// TIA Portal V18 export
FUNCTION_BLOCK "FB_MES_Monitoring"   // FB4, SCL
{ S7_Optimized_Access := 'TRUE' }
// stored: IsIECCheckEnabled true, MemoryReserve 100, SetENOAutomatically false
   VAR_INPUT
      Enable : Bool := TRUE;
      Reset : Bool := FALSE;
      HeartbeatTimeout_MES : Time := T#6s;
      HeartbeatTimeout_PLC : Time := T#6s;
      CheckInTimeout : Time := T#10s;
      CheckOutTimeout : Time := T#10s;
      StoveCheckInTimeout : Time := T#10s;
   END_VAR
   VAR_IN_OUT
      Diag : "UDT_MES_Monitoring";
   END_VAR
   VAR
      _hbMesValue : Bool;
      _hbPlcValue : Bool;
      _errCode : Array[1..8] of DInt;
      _errText : Array[1..8] of String[128];
      _actErrIdx : Array[1..8] of Int;
      _actErrCnt : Int;
      _actErrPos : Int;
      _errRotateEnable : Bool;
      _tErrRotate { S7_SetPoint := 'True'} : TON_TIME;
      _hbMesLast : Bool;
      _hbPlcLast : Bool;
      _tHbMes { S7_SetPoint := 'True'} : TON_TIME;
      _tHbPlc { S7_SetPoint := 'True'} : TON_TIME;
      _tCi { S7_SetPoint := 'True'} : Array[1..8] of TON_TIME;
      _tCo { S7_SetPoint := 'True'} : Array[1..8] of TON_TIME;
      _tStove { S7_SetPoint := 'True'} : TON_TIME;
      _ciDonePrev : Array[1..8] of Bool;
      _coDonePrev : Array[1..8] of Bool;
      _ciOkPrev : Array[1..8] of Bool;
      _ciNgPrev : Array[1..8] of Bool;
      _coOkPrev : Array[1..8] of Bool;
      _coNgPrev : Array[1..8] of Bool;
      _ciTimeoutLatched : Array[1..8] of Bool;
      _coTimeoutLatched : Array[1..8] of Bool;
      _spDonePrev : Array[1..8] of Bool;
      _spOkPrev : Array[1..8] of Bool;
      _spNgPrev : Array[1..8] of Bool;
      _lrDonePrev : Array[1..8] of Bool;
      _lrOkPrev : Array[1..8] of Bool;
      _lrNgPrev : Array[1..8] of Bool;
      _stoveOkPrev : Bool;
      _stoveTimeoutLatched : Bool;
      _i : Int;
      _ciReq : Array[1..8] of Bool;
      _ciOk : Array[1..8] of Bool;
      _ciNg : Array[1..8] of Bool;
      _ciDone : Array[1..8] of Bool;
      _coReq : Array[1..8] of Bool;
      _coOk : Array[1..8] of Bool;
      _coNg : Array[1..8] of Bool;
      _coDone : Array[1..8] of Bool;
      _spOk : Array[1..8] of Bool;
      _spNg : Array[1..8] of Bool;
      _spDone : Array[1..8] of Bool;
      _lrOk : Array[1..8] of Bool;
      _lrNg : Array[1..8] of Bool;
      _lrDone : Array[1..8] of Bool;
      _stoveReq : Bool;
      _stoveOk : Bool;
   END_VAR
BEGIN
   (*
   ===============================================================================
   BLOCK / PURPOSE
   ===============================================================================
   This code builds a MES diagnostics snapshot (#Diag) from PLC<->MES handshake DBs.
   It:
   - Mirrors key signals into #Diag.Header / #Diag.LastError / #Diag.Special / #Diag.Station[i]
   - Measures heartbeat "age" and timeout for MES and PLC heartbeats
   - Tracks per-station handshake counters (OK / NG / Done / Timeout) with edge detection
   - Latches "UnexpectedDone" if Done arrives without active request
   - Implements RESET to clear all counters/flags in #Diag
   ===============================================================================
   ASSUMPTIONS / NOTES
   ===============================================================================
   - #_tHbMes, #_tHbPlc, #_tStove and #_tCi[], #_tCo[] are IEC TON timers
   - #HeartbeatTimeout_MES / _PLC, #CheckInTimeout, #CheckOutTimeout, #StoveCheckInTimeout are TIME
   - Indexing: stations are 1..8
   - "ChickIn" naming in tags is preserved as-is (typo likely in original DB)
   ===============================================================================
   *)

   REGION "GUARD / ENABLE"
     IF NOT #Enable THEN
       RETURN;
     END_IF;
   END_REGION

   REGION "READ RAW SIGNALS FROM DBs (PLC<->MES + LAST ERROR)"
     #_hbMesValue := "MEStoPLC"."MES.HeartbeatSignal";
     #_hbPlcValue := "PLCtoMES"."PLC.Unload_HeartbeatSignal";

     // Unload error per station
     #_errCode[1] := "Station1UnLoadData"."MES.ErrorCode";
     #_errText[1] := "Station1UnLoadData"."MES.ErrorMsg";

     #_errCode[2] := "Station2UnLoadData"."MES.ErrorCode";
     #_errText[2] := "Station2UnLoadData"."MES.ErrorMsg";

     #_errCode[3] := "Station3UnLoadData"."MES.ErrorCode";
     #_errText[3] := "Station3UnLoadData"."MES.ErrorMsg";

     #_errCode[4] := "Station4UnLoadData"."MES.ErrorCode";
     #_errText[4] := "Station4UnLoadData"."MES.ErrorMsg";

     #_errCode[5] := "Station5UnLoadData"."MES.ErrorCode";
     #_errText[5] := "Station5UnLoadData"."MES.ErrorMsg";

     #_errCode[6] := "Station6UnLoadData"."MES.ErrorCode";
     #_errText[6] := "Station6UnLoadData"."MES.ErrorMsg";

     #_errCode[7] := "Station7UnLoadData"."MES.ErrorCode";
     #_errText[7] := "Station7UnLoadData"."MES.ErrorMsg";

     #_errCode[8] := "Station8UnLoadData"."MES.ErrorCode";
     #_errText[8] := "Station8UnLoadData"."MES.ErrorMsg";

     #_stoveReq := "PLCtoMES"."PLC.Load_StoveCheckIn";
     #_stoveOk := "MEStoPLC"."MES.Load_StoveCheckInOk";
   END_REGION


   REGION "MAP TO DIAG HEADER + LAST ERROR"
     #Diag.Header.Heartbeat_MES := #_hbMesValue;
     #Diag.Header.Heartbeat_PLC := #_hbPlcValue;

   END_REGION

   REGION "ACTIVE ERROR BUFFER + 3s ROTATE TO #Diag.LastError"
     // rebuild buffer each scan
     #_actErrCnt := 0;
     FOR #_i := 1 TO 8 DO
       // --- aktivni chyba kriterium ---
       IF (#_errCode[#_i] <> 0) THEN
         #_actErrCnt := #_actErrCnt + 1;
         #_actErrIdx[#_actErrCnt] := #_i;
       END_IF;
     END_FOR;

     // expose count to diag
     #Diag.LastError.ActCnt_Errors := #_actErrCnt;

     // keep pointer valid
     IF (#_actErrCnt = 0) THEN
       #_actErrPos := 1;
       #_errRotateEnable := FALSE;

       // when nothing active -> clear last error
       #Diag.LastError."Station Number" := 0;
       #Diag.LastError.Code := 0;
       #Diag.LastError.Text := '';
     ELSE
       IF (#_actErrPos < 1) OR (#_actErrPos > #_actErrCnt) THEN
         #_actErrPos := 1;
       END_IF;

       // start rotation timer if not running
       IF NOT #_errRotateEnable THEN
         #_errRotateEnable := TRUE;
       END_IF;

       // run 3s timer while enabled
       #_tErrRotate(IN := #_errRotateEnable,
                    PT := T#3S);

       // when 3s elapsed -> advance and force timer reset next scan
       IF #_tErrRotate.Q THEN
         #_errRotateEnable := FALSE;   // TON resets next scan (1-scan gap je OK)

         #_actErrPos := #_actErrPos + 1;
         IF #_actErrPos > #_actErrCnt THEN
           #_actErrPos := 1;
         END_IF;
       END_IF;

       // write currently selected active error to global LastError
       #_i := #_actErrIdx[#_actErrPos];   // reuse #_i jako index stanice (1..8)

       #Diag.LastError."Station Number" := #_i;
       #Diag.LastError.Code := #_errCode[#_i];

       // orez text do String[128] (kdyz DB ma delsi)
       #Diag.LastError.Text := LEFT(IN := #_errText[#_i], L := 128);
     END_IF;
   END_REGION

   REGION "HEARTBEAT SUPERVISION - MES -> PLC"
     // If heartbeat toggled since last scan => reset timer (forces ET back to 0)
     IF #_hbMesValue <> #_hbMesLast THEN
       #_hbMesLast := #_hbMesValue;
       #_tHbMes(IN := FALSE,
                PT := t#100ms);
     END_IF;

     // Run timer continuously; Q becomes TRUE after PT elapsed without heartbeat change
     #_tHbMes(IN := TRUE,
              PT := #HeartbeatTimeout_MES);

     #Diag.Header.MES_HeartbeatTimeout := #_tHbMes.Q;   // TRUE = timeout reached
     #Diag.Header.MES_HeartbeatAge := #_tHbMes.ET;  // elapsed since last toggle
     #Diag.Header.MES_Online := NOT #_tHbMes.Q;
   END_REGION


   REGION "HEARTBEAT SUPERVISION - PLC -> MES"
     // If heartbeat toggled => reset PLC heartbeat timer
     IF #_hbPlcValue <> #_hbPlcLast THEN
       #_hbPlcLast := #_hbPlcValue;
       #_tHbPlc(IN := FALSE,
                PT := t#100ms);
     END_IF;

     // Run timer continuously
     #_tHbPlc(IN := TRUE,
              PT := #HeartbeatTimeout_PLC);

     #Diag.Header.PLC_HeartbeatTimeout := #_tHbPlc.Q;
     #Diag.Header.PLC_HeartbeatAge := #_tHbPlc.ET;
   END_REGION


   REGION "BUILD HANDSHAKE ARRAYS (READ INPUTS ONCE) - CHECK-IN REQ/OK/NG/DONE"
     // Check-in request bits (PLC -> MES), one per station
     #_ciReq[1] := "PLCtoMES"."PLC.Load_Station1ChickInReq";
     #_ciReq[2] := "PLCtoMES"."PLC.Load_Station2ChickInReq";
     #_ciReq[3] := "PLCtoMES"."PLC.Load_Station3ChickInReq";
     #_ciReq[4] := "PLCtoMES"."PLC.Load_Station4ChickInReq";
     #_ciReq[5] := "PLCtoMES"."PLC.Load_Station5ChickInReq";
     #_ciReq[6] := "PLCtoMES"."PLC.Load_Station6ChickInReq";
     #_ciReq[7] := "PLCtoMES"."PLC.Load_Station7ChickInReq";
     #_ciReq[8] := "PLCtoMES"."PLC.Load_Station8ChickInReq";

     // Check-in result bits from MES (OK / NG / Done)
     #_ciOk[1] := "MEStoPLC"."MES.Load_Station1PartOK";
     #_ciOk[2] := "MEStoPLC"."MES.Load_Station2PartOK";
     #_ciOk[3] := "MEStoPLC"."MES.Load_Station3PartOK";
     #_ciOk[4] := "MEStoPLC"."MES.Load_Station4PartOK";
     #_ciOk[5] := "MEStoPLC"."MES.Load_Station5PartOK";
     #_ciOk[6] := "MEStoPLC"."MES.Load_Station6PartOK";
     #_ciOk[7] := "MEStoPLC"."MES.Load_Station7PartOK";
     #_ciOk[8] := "MEStoPLC"."MES.Load_Station8PartOK";

     #_ciNg[1] := "MEStoPLC"."MES.Load_Station1PartNG";
     #_ciNg[2] := "MEStoPLC"."MES.Load_Station2PartNG";
     #_ciNg[3] := "MEStoPLC"."MES.Load_Station3PartNG";
     #_ciNg[4] := "MEStoPLC"."MES.Load_Station4PartNG";
     #_ciNg[5] := "MEStoPLC"."MES.Load_Station5PartNG";
     #_ciNg[6] := "MEStoPLC"."MES.Load_Station6PartNG";
     #_ciNg[7] := "MEStoPLC"."MES.Load_Station7PartNG";
     #_ciNg[8] := "MEStoPLC"."MES.Load_Station8PartNG";

     #_ciDone[1] := "MEStoPLC"."MES.Load_Station1ReqMesDone";
     #_ciDone[2] := "MEStoPLC"."MES.Load_Station2ReqMesDone";
     #_ciDone[3] := "MEStoPLC"."MES.Load_Station3ReqMesDone";
     #_ciDone[4] := "MEStoPLC"."MES.Load_Station4ReqMesDone";
     #_ciDone[5] := "MEStoPLC"."MES.Load_Station5ReqMesDone";
     #_ciDone[6] := "MEStoPLC"."MES.Load_Station6ReqMesDone";
     #_ciDone[7] := "MEStoPLC"."MES.Load_Station7ReqMesDone";
     #_ciDone[8] := "MEStoPLC"."MES.Load_Station8ReqMesDone";
   END_REGION


   REGION "BUILD HANDSHAKE ARRAYS (READ INPUTS ONCE) - CHECK-OUT REQ/OK/NG/DONE"
     // Check-out request bits (PLC -> MES): request to save unload data
     #_coReq[1] := "PLCtoMES"."PLC.Unload_Station1DataSaveReq";
     #_coReq[2] := "PLCtoMES"."PLC.Unload_Station2DataSaveReq";
     #_coReq[3] := "PLCtoMES"."PLC.Unload_Station3DataSaveReq";
     #_coReq[4] := "PLCtoMES"."PLC.Unload_Station4DataSaveReq";
     #_coReq[5] := "PLCtoMES"."PLC.Unload_Station5DataSaveReq";
     #_coReq[6] := "PLCtoMES"."PLC.Unload_Station6DataSaveReq";
     #_coReq[7] := "PLCtoMES"."PLC.Unload_Station7DataSaveReq";
     #_coReq[8] := "PLCtoMES"."PLC.Unload_Station8DataSaveReq";

     // Check-out results (OK/NG/Done) from MES
     #_coOk[1] := "MEStoPLC"."MES.Unload_ResultsStored1OK";
     #_coOk[2] := "MEStoPLC"."MES.Unload_ResultsStored2OK";
     #_coOk[3] := "MEStoPLC"."MES.Unload_ResultsStored3OK";
     #_coOk[4] := "MEStoPLC"."MES.Unload_ResultsStored4OK";
     #_coOk[5] := "MEStoPLC"."MES.Unload_ResultsStored5OK";
     #_coOk[6] := "MEStoPLC"."MES.Unload_ResultsStored6OK";
     #_coOk[7] := "MEStoPLC"."MES.Unload_ResultsStored7OK";
     #_coOk[8] := "MEStoPLC"."MES.Unload_ResultsStored8OK";

     #_coNg[1] := "MEStoPLC"."MES.Unload_ResultsStored1NG";
     #_coNg[2] := "MEStoPLC"."MES.Unload_ResultsStored2NG";
     #_coNg[3] := "MEStoPLC"."MES.Unload_ResultsStored3NG";
     #_coNg[4] := "MEStoPLC"."MES.Unload_ResultsStored4NG";
     #_coNg[5] := "MEStoPLC"."MES.Unload_ResultsStored5NG";
     #_coNg[6] := "MEStoPLC"."MES.Unload_ResultsStored6NG";
     #_coNg[7] := "MEStoPLC"."MES.Unload_ResultsStored7NG";
     #_coNg[8] := "MEStoPLC"."MES.Unload_ResultsStored8NG";

     #_coDone[1] := "MEStoPLC"."MES.Unload_ResultsStored1ReqMesDone";
     #_coDone[2] := "MEStoPLC"."MES.Unload_ResultsStored2ReqMesDone";
     #_coDone[3] := "MEStoPLC"."MES.Unload_ResultsStored3ReqMesDone";
     #_coDone[4] := "MEStoPLC"."MES.Unload_ResultsStored4ReqMesDone";
     #_coDone[5] := "MEStoPLC"."MES.Unload_ResultsStored5ReqMesDone";
     #_coDone[6] := "MEStoPLC"."MES.Unload_ResultsStored6ReqMesDone";
     #_coDone[7] := "MEStoPLC"."MES.Unload_ResultsStored7ReqMesDone";
     #_coDone[8] := "MEStoPLC"."MES.Unload_ResultsStored8ReqMesDone";
   END_REGION


   REGION "BUILD HANDSHAKE ARRAYS - SUBPART OK/NG/DONE (LOAD SIDE)"
     #_spOk[1] := "MEStoPLC"."MES.Load_SubPart1OK";
     #_spOk[2] := "MEStoPLC"."MES.Load_SubPart2OK";
     #_spOk[3] := "MEStoPLC"."MES.Load_SubPart3OK";
     #_spOk[4] := "MEStoPLC"."MES.Load_SubPart4OK";
     #_spOk[5] := "MEStoPLC"."MES.Load_SubPart5OK";
     #_spOk[6] := "MEStoPLC"."MES.Load_SubPart6OK";
     #_spOk[7] := "MEStoPLC"."MES.Load_SubPart7OK";
     #_spOk[8] := "MEStoPLC"."MES.Load_SubPart8OK";

     // NOTE: tags contain "...SubPartXtNG" (typo) - preserved exactly as given
     #_spNg[1] := "MEStoPLC"."MES.Load_SubPart1tNG";
     #_spNg[2] := "MEStoPLC"."MES.Load_SubPart2tNG";
     #_spNg[3] := "MEStoPLC"."MES.Load_SubPart3tNG";
     #_spNg[4] := "MEStoPLC"."MES.Load_SubPart4tNG";
     #_spNg[5] := "MEStoPLC"."MES.Load_SubPart5tNG";
     #_spNg[6] := "MEStoPLC"."MES.Load_SubPart6tNG";
     #_spNg[7] := "MEStoPLC"."MES.Load_SubPart7tNG";
     #_spNg[8] := "MEStoPLC"."MES.Load_SubPart8tNG";

     #_spDone[1] := "MEStoPLC"."MES.Load_SubPart1ReqMesDone";
     #_spDone[2] := "MEStoPLC"."MES.Load_SubPart2ReqMesDone";
     #_spDone[3] := "MEStoPLC"."MES.Load_SubPart3ReqMesDone";
     #_spDone[4] := "MEStoPLC"."MES.Load_SubPart4ReqMesDone";
     #_spDone[5] := "MEStoPLC"."MES.Load_SubPart5ReqMesDone";
     #_spDone[6] := "MEStoPLC"."MES.Load_SubPart6ReqMesDone";
     #_spDone[7] := "MEStoPLC"."MES.Load_SubPart7ReqMesDone";
     #_spDone[8] := "MEStoPLC"."MES.Load_SubPart8ReqMesDone";
   END_REGION


   REGION "BUILD HANDSHAKE ARRAYS - LOAD RESULTS STORED OK/NG/DONE (LOAD SIDE)"
     #_lrOk[1] := "MEStoPLC"."MES.Load_ResultsStored1OK";
     #_lrOk[2] := "MEStoPLC"."MES.Load_ResultsStored2OK";
     #_lrOk[3] := "MEStoPLC"."MES.Load_ResultsStored3OK";
     #_lrOk[4] := "MEStoPLC"."MES.Load_ResultsStored4OK";
     #_lrOk[5] := "MEStoPLC"."MES.Load_ResultsStored5OK";
     #_lrOk[6] := "MEStoPLC"."MES.Load_ResultsStored6OK";
     #_lrOk[7] := "MEStoPLC"."MES.Load_ResultsStored7OK";
     #_lrOk[8] := "MEStoPLC"."MES.Load_ResultsStored8OK";

     #_lrNg[1] := "MEStoPLC"."MES.Load_ResultsStored1NG";
     #_lrNg[2] := "MEStoPLC"."MES.Load_ResultsStored2NG";
     #_lrNg[3] := "MEStoPLC"."MES.Load_ResultsStored3NG";
     #_lrNg[4] := "MEStoPLC"."MES.Load_ResultsStored4NG";
     #_lrNg[5] := "MEStoPLC"."MES.Load_ResultsStored5NG";
     #_lrNg[6] := "MEStoPLC"."MES.Load_ResultsStored6NG";
     #_lrNg[7] := "MEStoPLC"."MES.Load_ResultsStored7NG";
     #_lrNg[8] := "MEStoPLC"."MES.Load_ResultsStored8NG";

     #_lrDone[1] := "MEStoPLC"."MES.Load_ResultsStored1ReqMesDone";
     #_lrDone[2] := "MEStoPLC"."MES.Load_ResultsStored2ReqMesDone";
     #_lrDone[3] := "MEStoPLC"."MES.Load_ResultsStored3ReqMesDone";
     #_lrDone[4] := "MEStoPLC"."MES.Load_ResultsStored4ReqMesDone";
     #_lrDone[5] := "MEStoPLC"."MES.Load_ResultsStored5ReqMesDone";
     #_lrDone[6] := "MEStoPLC"."MES.Load_ResultsStored6ReqMesDone";
     #_lrDone[7] := "MEStoPLC"."MES.Load_ResultsStored7ReqMesDone";
     #_lrDone[8] := "MEStoPLC"."MES.Load_ResultsStored8ReqMesDone";
   END_REGION


   REGION "RESET DIAGNOSTICS (COUNTERS + LATCHES)"
     IF #Reset THEN
       FOR #_i := 1 TO 8 DO
         // Station-level latches
         #Diag.Station[#_i].CheckIn.UnexpectedDone := FALSE;
         #Diag.Station[#_i].CheckOut.UnexpectedDone := FALSE;

         // Per-station counters: SubPart
         #Diag.Station[#_i].SubPart.CountOK := 0;
         #Diag.Station[#_i].SubPart.CountNG := 0;
         #Diag.Station[#_i].SubPart.CountDone := 0;

         // Per-station counters: LoadResultsStored
         #Diag.Station[#_i].LoadResultsStored.CountOK := 0;
         #Diag.Station[#_i].LoadResultsStored.CountNG := 0;
         #Diag.Station[#_i].LoadResultsStored.CountDone := 0;

         // Per-station counters: CheckIn
         #Diag.Station[#_i].CheckIn.CountOK := 0;
         #Diag.Station[#_i].CheckIn.CountNG := 0;
         #Diag.Station[#_i].CheckIn.CountDone := 0;
         #Diag.Station[#_i].CheckIn.CountTimeout := 0;

         // Per-station counters: CheckOut
         #Diag.Station[#_i].CheckOut.CountOK := 0;
         #Diag.Station[#_i].CheckOut.CountNG := 0;
         #Diag.Station[#_i].CheckOut.CountDone := 0;
         #Diag.Station[#_i].CheckOut.CountTimeout := 0;

         // Internal timeout latch states (avoid re-counting while timeout stays TRUE)
         #_ciTimeoutLatched[#_i] := FALSE;
         #_coTimeoutLatched[#_i] := FALSE;
       END_FOR;

       // Special (stove) counters / latches
       #Diag.Special.CountOk := 0;
       #Diag.Special.CountTimeout := 0;
       #_stoveTimeoutLatched := FALSE;
     END_IF;
   END_REGION


   REGION "RESET TOTAL COUNTERS (RE-CALCULATED EACH SCAN)"
     #Diag.Counters.TotalDone_CheckIn := 0;
     #Diag.Counters.TotalDone_CheckOut := 0;
     #Diag.Counters.TotalTimeout_CheckIn := 0;
     #Diag.Counters.TotalTimeout_CheckOut := 0;
     #Diag.Counters.TotalOK_CheckIn := 0;
     #Diag.Counters.TotalNG_CheckIn := 0;
     #Diag.Counters.TotalOK_CheckOut := 0;
     #Diag.Counters.TotalNG_CheckOut := 0;
   END_REGION


   REGION "MAIN LOOP 1..8 - STATION DIAGNOSTICS + EDGE COUNTERS + TIMEOUTS"
     FOR #_i := 1 TO 8 DO


       REGION "MAP STATION DATA (LOAD/UNLOAD) -> Diag.Station[i].*.DATA"
         // konstanta cisla stanice do Diag (pokud mas v UDT StationNumber)

         CASE #_i OF

           1:
             // ================== LOAD: Station1LoadData ==================
             #Diag.Station[#_i].CheckIn.DATA.PLC_PartTypeID := "Station1LoadData"."PLC.PartTypeID";
             #Diag.Station[#_i].CheckIn.DATA.PLC_StationRecipeNo := "Station1LoadData"."PLC.Station1RecipeNo";
             #Diag.Station[#_i].CheckIn.DATA.PLC_StationDMXCode := "Station1LoadData"."PLC.Station1DMXCode";
             #Diag.Station[#_i].CheckIn.DATA.PLC_StationStatus := "Station1LoadData"."PLC.StationStatus";
             #Diag.Station[#_i].CheckIn.DATA.MES_ErrorCode := "Station1LoadData"."MES.ErrorCode";
             #Diag.Station[#_i].CheckIn.DATA.MES_StatusBits := "Station1LoadData"."MES.StatusBits";
             #Diag.Station[#_i].CheckIn.DATA.MES_Cycle_ID := "Station1LoadData"."MES.Cycle_ID";
             #Diag.Station[#_i].CheckIn.DATA.MES_Unit_ParttypeID := "Station1LoadData"."MES.Unit_ParttypeID";

             // ================== UNLOAD: Station1UnLoadData ==================
             #Diag.Station[#_i].CheckOut.DATA.PLC_PartTypeID := "Station1UnLoadData"."PLC.PartTypeID";
             #Diag.Station[#_i].CheckOut.DATA.PLC_StationDMXCode := "Station1UnLoadData"."PLC.Station1DMXCode";
             #Diag.Station[#_i].CheckOut.DATA.PLC_StationRecipeNo := "Station1UnLoadData"."PLC.Station1RecipeNo";
             #Diag.Station[#_i].CheckOut.DATA.PLC_PartStatus := "Station1UnLoadData"."PLC.PartStatus";
             #Diag.Station[#_i].CheckOut.DATA.PLC_SubPartSN1 := "Station1UnLoadData"."PLC.SubPartSN1";
             #Diag.Station[#_i].CheckOut.DATA.PLC_TransferTime := "Station1UnLoadData"."PLC.TransferTime";
           //  #Diag.Station[#_i].CheckOut.DATA."PLC.NGCode" := "Station1UnLoadData"."PLC.NGCode";
             #Diag.Station[#_i].CheckOut.DATA.MES_ErrorCode := "Station1UnLoadData"."MES.ErrorCode";
             #Diag.Station[#_i].CheckOut.DATA.MES_ErrorMsg := "Station1UnLoadData"."MES.ErrorMsg";

           2:
             #Diag.Station[#_i].CheckIn.DATA.PLC_PartTypeID := "Station2LoadData"."PLC.PartTypeID";
             #Diag.Station[#_i].CheckIn.DATA.PLC_StationRecipeNo := "Station2LoadData"."PLC.Station2RecipeNo";
             #Diag.Station[#_i].CheckIn.DATA.PLC_StationDMXCode := "Station2LoadData"."PLC.Station2DMXCode";
          //   #Diag.Station[#_i].CheckIn.DATA."PLC.StationStatus" := "Station2LoadData"."PLC.StationStatus";
             #Diag.Station[#_i].CheckIn.DATA.MES_ErrorCode := "Station2LoadData"."MES.ErrorCode";
             #Diag.Station[#_i].CheckIn.DATA.MES_StatusBits := "Station2LoadData"."MES.StatusBits";
             #Diag.Station[#_i].CheckIn.DATA.MES_Cycle_ID := "Station2LoadData"."MES.Cycle_ID";
             #Diag.Station[#_i].CheckIn.DATA.MES_Unit_ParttypeID := "Station2LoadData"."MES.Unit_ParttypeID";

             #Diag.Station[#_i].CheckOut.DATA.PLC_PartTypeID := "Station2UnLoadData"."PLC.PartTypeID";
             #Diag.Station[#_i].CheckOut.DATA.PLC_StationDMXCode := "Station2UnLoadData"."PLC.Station2DMXCode";
             #Diag.Station[#_i].CheckOut.DATA.PLC_StationRecipeNo := "Station2UnLoadData"."PLC.Station2RecipeNo";
             #Diag.Station[#_i].CheckOut.DATA.PLC_PartStatus := "Station2UnLoadData"."PLC.PartStatus";
             #Diag.Station[#_i].CheckOut.DATA.PLC_SubPartSN1 := "Station2UnLoadData"."PLC.SubPartSN1";
             #Diag.Station[#_i].CheckOut.DATA.PLC_TransferTime := "Station2UnLoadData"."PLC.TransferTime";
         //    #Diag.Station[#_i].CheckOut.DATA."PLC.NGCode" := "Station2UnLoadData"."PLC.NGCode";
             #Diag.Station[#_i].CheckOut.DATA.MES_ErrorCode := "Station2UnLoadData"."MES.ErrorCode";
             #Diag.Station[#_i].CheckOut.DATA.MES_ErrorMsg := "Station2UnLoadData"."MES.ErrorMsg";

           3:
             #Diag.Station[#_i].CheckIn.DATA.PLC_PartTypeID := "Station3LoadData"."PLC.PartTypeID";
             #Diag.Station[#_i].CheckIn.DATA.PLC_StationRecipeNo := "Station3LoadData"."PLC.Station3RecipeNo";
             #Diag.Station[#_i].CheckIn.DATA.PLC_StationDMXCode := "Station3LoadData"."PLC.Station3DMXCode";
         //    #Diag.Station[#_i].CheckIn.DATA."PLC.StationStatus" := "Station3LoadData"."PLC.StationStatus";
             #Diag.Station[#_i].CheckIn.DATA.MES_ErrorCode := "Station3LoadData"."MES.ErrorCode";
             #Diag.Station[#_i].CheckIn.DATA.MES_StatusBits := "Station3LoadData"."MES.StatusBits";
             #Diag.Station[#_i].CheckIn.DATA.MES_Cycle_ID := "Station3LoadData"."MES.Cycle_ID";
             #Diag.Station[#_i].CheckIn.DATA.MES_Unit_ParttypeID := "Station3LoadData"."MES.Unit_ParttypeID";

             #Diag.Station[#_i].CheckOut.DATA.PLC_PartTypeID := "Station3UnLoadData"."PLC.PartTypeID";
             #Diag.Station[#_i].CheckOut.DATA.PLC_StationDMXCode := "Station3UnLoadData"."PLC.Station3DMXCode";
             #Diag.Station[#_i].CheckOut.DATA.PLC_StationRecipeNo := "Station3UnLoadData"."PLC.Station3RecipeNo";
             #Diag.Station[#_i].CheckOut.DATA.PLC_PartStatus := "Station3UnLoadData"."PLC.PartStatus";
             #Diag.Station[#_i].CheckOut.DATA.PLC_SubPartSN1 := "Station3UnLoadData"."PLC.SubPartSN1";
             #Diag.Station[#_i].CheckOut.DATA.PLC_TransferTime := "Station3UnLoadData"."PLC.TransferTime";
             #Diag.Station[#_i].CheckOut.DATA.PLC_NGCode := "Station3UnLoadData"."PLC.NGCode";
             #Diag.Station[#_i].CheckOut.DATA.MES_ErrorCode := "Station3UnLoadData"."MES.ErrorCode";
             #Diag.Station[#_i].CheckOut.DATA.MES_ErrorMsg := "Station3UnLoadData"."MES.ErrorMsg";

           4:
             #Diag.Station[#_i].CheckIn.DATA.PLC_PartTypeID := "Station4LoadData"."PLC.PartTypeID";
             #Diag.Station[#_i].CheckIn.DATA.PLC_StationRecipeNo := "Station4LoadData"."PLC.Station4RecipeNo";
             #Diag.Station[#_i].CheckIn.DATA.PLC_StationDMXCode := "Station4LoadData"."PLC.Station4DMXCode";
           //  #Diag.Station[#_i].CheckIn.DATA."PLC.StationStatus" := "Station4LoadData"."PLC.StationStatus";
             #Diag.Station[#_i].CheckIn.DATA.MES_ErrorCode := "Station4LoadData"."MES.ErrorCode";
             #Diag.Station[#_i].CheckIn.DATA.MES_StatusBits := "Station4LoadData"."MES.StatusBits";
             #Diag.Station[#_i].CheckIn.DATA.MES_Cycle_ID := "Station4LoadData"."MES.Cycle_ID";
             #Diag.Station[#_i].CheckIn.DATA.MES_Unit_ParttypeID := "Station4LoadData"."MES.Unit_ParttypeID";

             #Diag.Station[#_i].CheckOut.DATA.PLC_PartTypeID := "Station4UnLoadData"."PLC.PartTypeID";
             #Diag.Station[#_i].CheckOut.DATA.PLC_StationDMXCode := "Station4UnLoadData"."PLC.Station4DMXCode";
             #Diag.Station[#_i].CheckOut.DATA.PLC_StationRecipeNo := "Station4UnLoadData"."PLC.Station4RecipeNo";
             #Diag.Station[#_i].CheckOut.DATA.PLC_PartStatus := "Station4UnLoadData"."PLC.PartStatus";
             #Diag.Station[#_i].CheckOut.DATA.PLC_SubPartSN1 := "Station4UnLoadData"."PLC.SubPartSN1";
             #Diag.Station[#_i].CheckOut.DATA.PLC_TransferTime := "Station4UnLoadData"."PLC.TransferTime";
         //    #Diag.Station[#_i].CheckOut.DATA."PLC.NGCode" := "Station4UnLoadData"."PLC.NGCode";
             #Diag.Station[#_i].CheckOut.DATA.MES_ErrorCode := "Station4UnLoadData"."MES.ErrorCode";
             #Diag.Station[#_i].CheckOut.DATA.MES_ErrorMsg := "Station4UnLoadData"."MES.ErrorMsg";

           5:
             #Diag.Station[#_i].CheckIn.DATA.PLC_PartTypeID := "Station5LoadData"."PLC.PartTypeID";
             #Diag.Station[#_i].CheckIn.DATA.PLC_StationRecipeNo := "Station5LoadData"."PLC.Station5RecipeNo";
             #Diag.Station[#_i].CheckIn.DATA.PLC_StationDMXCode := "Station5LoadData"."PLC.Station5DMXCode";
        //     #Diag.Station[#_i].CheckIn.DATA."PLC.StationStatus" := "Station5LoadData"."PLC.StationStatus";
             #Diag.Station[#_i].CheckIn.DATA.MES_ErrorCode := "Station5LoadData"."MES.ErrorCode";
             #Diag.Station[#_i].CheckIn.DATA.MES_StatusBits := "Station5LoadData"."MES.StatusBits";
             #Diag.Station[#_i].CheckIn.DATA.MES_Cycle_ID := "Station5LoadData"."MES.Cycle_ID";
             #Diag.Station[#_i].CheckIn.DATA.MES_Unit_ParttypeID := "Station5LoadData"."MES.Unit_ParttypeID";

             #Diag.Station[#_i].CheckOut.DATA.PLC_PartTypeID := "Station5UnLoadData"."PLC.PartTypeID";
             #Diag.Station[#_i].CheckOut.DATA.PLC_StationDMXCode := "Station5UnLoadData"."PLC.Station5DMXCode";
             #Diag.Station[#_i].CheckOut.DATA.PLC_StationRecipeNo := "Station5UnLoadData"."PLC.Station5RecipeNo";
             #Diag.Station[#_i].CheckOut.DATA.PLC_PartStatus := "Station5UnLoadData"."PLC.PartStatus";
             #Diag.Station[#_i].CheckOut.DATA.PLC_SubPartSN1 := "Station5UnLoadData"."PLC.SubPartSN1";
             #Diag.Station[#_i].CheckOut.DATA.PLC_TransferTime := "Station5UnLoadData"."PLC.TransferTime";
             #Diag.Station[#_i].CheckOut.DATA.PLC_NGCode := "Station5UnLoadData"."PLC.NGCode";
             #Diag.Station[#_i].CheckOut.DATA.MES_ErrorCode := "Station5UnLoadData"."MES.ErrorCode";
             #Diag.Station[#_i].CheckOut.DATA.MES_ErrorMsg := "Station5UnLoadData"."MES.ErrorMsg";

           6:
             #Diag.Station[#_i].CheckIn.DATA.PLC_PartTypeID := "Station6LoadData"."PLC.PartTypeID";
             #Diag.Station[#_i].CheckIn.DATA.PLC_StationRecipeNo := "Station6LoadData"."PLC.Station6RecipeNo";
             #Diag.Station[#_i].CheckIn.DATA.PLC_StationDMXCode := "Station6LoadData"."PLC.Station6DMXCode";
         //    #Diag.Station[#_i].CheckIn.DATA."PLC.StationStatus" := "Station6LoadData"."PLC.StationStatus";
             #Diag.Station[#_i].CheckIn.DATA.MES_ErrorCode := "Station6LoadData"."MES.ErrorCode";
             #Diag.Station[#_i].CheckIn.DATA.MES_StatusBits := "Station6LoadData"."MES.StatusBits";
             #Diag.Station[#_i].CheckIn.DATA.MES_Cycle_ID := "Station6LoadData"."MES.Cycle_ID";
             #Diag.Station[#_i].CheckIn.DATA.MES_Unit_ParttypeID := "Station6LoadData"."MES.Unit_ParttypeID";

             #Diag.Station[#_i].CheckOut.DATA.PLC_PartTypeID := "Station6UnLoadData"."PLC.PartTypeID";
             #Diag.Station[#_i].CheckOut.DATA.PLC_StationDMXCode := "Station6UnLoadData"."PLC.Station6DMXCode";
             #Diag.Station[#_i].CheckOut.DATA.PLC_StationRecipeNo := "Station6UnLoadData"."PLC.Station6RecipeNo";
             #Diag.Station[#_i].CheckOut.DATA.PLC_PartStatus := "Station6UnLoadData"."PLC.PartStatus";
             #Diag.Station[#_i].CheckOut.DATA.PLC_SubPartSN1 := "Station6UnLoadData"."PLC.SubPartSN1";
             #Diag.Station[#_i].CheckOut.DATA.PLC_TransferTime := "Station6UnLoadData"."PLC.TransferTime";
         //    #Diag.Station[#_i].CheckOut.DATA."PLC.NGCode" := "Station6UnLoadData"."PLC.NGCode";
             #Diag.Station[#_i].CheckOut.DATA.MES_ErrorCode := "Station6UnLoadData"."MES.ErrorCode";
             #Diag.Station[#_i].CheckOut.DATA.MES_ErrorMsg := "Station6UnLoadData"."MES.ErrorMsg";

           7:
             #Diag.Station[#_i].CheckIn.DATA.PLC_PartTypeID := "Station7LoadData"."PLC.PartTypeID";
             #Diag.Station[#_i].CheckIn.DATA.PLC_StationRecipeNo := "Station7LoadData"."PLC.Station7RecipeNo";
             #Diag.Station[#_i].CheckIn.DATA.PLC_StationDMXCode := "Station7LoadData"."PLC.Station7DMXCode";
     //        #Diag.Station[#_i].CheckIn.DATA."PLC.StationStatus" := "Station7LoadData"."PLC.StationStatus";
             #Diag.Station[#_i].CheckIn.DATA.MES_ErrorCode := "Station7LoadData"."MES.ErrorCode";
             #Diag.Station[#_i].CheckIn.DATA.MES_StatusBits := "Station7LoadData"."MES.StatusBits";
             #Diag.Station[#_i].CheckIn.DATA.MES_Cycle_ID := "Station7LoadData"."MES.Cycle_ID";
             #Diag.Station[#_i].CheckIn.DATA.MES_Unit_ParttypeID := "Station7LoadData"."MES.Unit_ParttypeID";

             #Diag.Station[#_i].CheckOut.DATA.PLC_PartTypeID := "Station7UnLoadData"."PLC.PartTypeID";
             #Diag.Station[#_i].CheckOut.DATA.PLC_StationDMXCode := "Station7UnLoadData"."PLC.Station7DMXCode";
             #Diag.Station[#_i].CheckOut.DATA.PLC_StationRecipeNo := "Station7UnLoadData"."PLC.Station7RecipeNo";
             #Diag.Station[#_i].CheckOut.DATA.PLC_PartStatus := "Station7UnLoadData"."PLC.PartStatus";
             #Diag.Station[#_i].CheckOut.DATA.PLC_SubPartSN1 := "Station7UnLoadData"."PLC.SubPartSN1";
             #Diag.Station[#_i].CheckOut.DATA.PLC_TransferTime := "Station7UnLoadData"."PLC.TransferTime";
             #Diag.Station[#_i].CheckOut.DATA.PLC_NGCode := "Station7UnLoadData"."PLC.NGCode";
             #Diag.Station[#_i].CheckOut.DATA.MES_ErrorCode := "Station7UnLoadData"."MES.ErrorCode";
             #Diag.Station[#_i].CheckOut.DATA.MES_ErrorMsg := "Station7UnLoadData"."MES.ErrorMsg";

           8:
             #Diag.Station[#_i].CheckIn.DATA.PLC_PartTypeID := "Station8LoadData"."PLC.PartTypeID";
             #Diag.Station[#_i].CheckIn.DATA.PLC_StationRecipeNo := "Station8LoadData"."PLC.Station8RecipeNo";
             #Diag.Station[#_i].CheckIn.DATA.PLC_StationDMXCode := "Station8LoadData"."PLC.Station8DMXCode";
   //          #Diag.Station[#_i].CheckIn.DATA."PLC.StationStatus" := "Station8LoadData"."PLC.StationStatus";
             #Diag.Station[#_i].CheckIn.DATA.MES_ErrorCode := "Station8LoadData"."MES.ErrorCode";
             #Diag.Station[#_i].CheckIn.DATA.MES_StatusBits := "Station8LoadData"."MES.StatusBits";
             #Diag.Station[#_i].CheckIn.DATA.MES_Cycle_ID := "Station8LoadData"."MES.Cycle_ID";
             #Diag.Station[#_i].CheckIn.DATA.MES_Unit_ParttypeID := "Station8LoadData"."MES.Unit_ParttypeID";

             #Diag.Station[#_i].CheckOut.DATA.PLC_PartTypeID := "Station8UnLoadData"."PLC.PartTypeID";
        //     #Diag.Station[#_i].CheckOut.DATA."PLC.StationDMXCode" := "Station8UnLoadData"."PLC.Station8DMXCode";
       //      #Diag.Station[#_i].CheckOut.DATA."PLC.StationRecipeNo" := "Station8UnLoadData"."PLC.Station8RecipeNo";
             #Diag.Station[#_i].CheckOut.DATA.PLC_PartStatus := "Station8UnLoadData"."PLC.PartStatus";
             #Diag.Station[#_i].CheckOut.DATA.PLC_SubPartSN1 := "Station8UnLoadData"."PLC.SubPartSN1";
             #Diag.Station[#_i].CheckOut.DATA.PLC_TransferTime := "Station8UnLoadData"."PLC.TransferTime";
       //      #Diag.Station[#_i].CheckOut.DATA."PLC.NGCode" := "Station8UnLoadData"."PLC.NGCode";
             #Diag.Station[#_i].CheckOut.DATA.MES_ErrorCode := "Station8UnLoadData"."MES.ErrorCode";
             #Diag.Station[#_i].CheckOut.DATA.MES_ErrorMsg := "Station8UnLoadData"."MES.ErrorMsg";

         END_CASE;
       END_REGION


       // --------------------------------------------------------------------------
       // CHECK-IN DIAG (Load)
       // --------------------------------------------------------------------------
       #Diag.Station[#_i].CheckIn.Req := #_ciReq[#_i];
       #Diag.Station[#_i].CheckIn.OK := #_ciOk[#_i];
       #Diag.Station[#_i].CheckIn.NG := #_ciNg[#_i];
       #Diag.Station[#_i].CheckIn.Done := #_ciDone[#_i];

       // Invalid state detector: OK and NG simultaneously
       #Diag.Station[#_i].CheckIn.BothOkNg := #_ciOk[#_i] AND #_ciNg[#_i];

       // Rising edge count: OK
       IF #_ciOk[#_i] AND (NOT #_ciOkPrev[#_i]) THEN
         #Diag.Station[#_i].CheckIn.CountOK := #Diag.Station[#_i].CheckIn.CountOK + 1;
       END_IF;
       #_ciOkPrev[#_i] := #_ciOk[#_i];

       // Rising edge count: NG
       IF #_ciNg[#_i] AND (NOT #_ciNgPrev[#_i]) THEN
         #Diag.Station[#_i].CheckIn.CountNG := #Diag.Station[#_i].CheckIn.CountNG + 1;
       END_IF;
       #_ciNgPrev[#_i] := #_ciNg[#_i];

       // Timer: measure duration of active request
       IF #_ciReq[#_i] THEN
         #_tCi[#_i](IN := TRUE,
                    PT := #CheckInTimeout);
         #Diag.Station[#_i].CheckIn.InProgress := TRUE;
       ELSE
         // Reset timer when request is inactive
         #_tCi[#_i](IN := FALSE,
                    PT := t#100ms);
         #Diag.Station[#_i].CheckIn.InProgress := FALSE;
       END_IF;

       #Diag.Station[#_i].CheckIn.Elapsed := #_tCi[#_i].ET;

       // Timeout: timer expired while request still active and Done not received
       #Diag.Station[#_i].CheckIn.Timeout :=
       #_tCi[#_i].Q AND #_ciReq[#_i] AND (NOT #_ciDone[#_i]);

       // Count timeout only on first scan of timeout assertion (latch)
       IF #Diag.Station[#_i].CheckIn.Timeout AND (NOT #_ciTimeoutLatched[#_i]) THEN
         #_ciTimeoutLatched[#_i] := TRUE;
         #Diag.Station[#_i].CheckIn.CountTimeout := #Diag.Station[#_i].CheckIn.CountTimeout + 1;
       END_IF;

       // Release latch when timeout condition clears
       IF NOT #Diag.Station[#_i].CheckIn.Timeout THEN
         #_ciTimeoutLatched[#_i] := FALSE;
       END_IF;

       // Rising edge count: Done + UnexpectedDone latch if no active request
       IF #_ciDone[#_i] AND (NOT #_ciDonePrev[#_i]) THEN
         #Diag.Station[#_i].CheckIn.CountDone := #Diag.Station[#_i].CheckIn.CountDone + 1;

         // Done without request: indicates inconsistent handshake timing or stale signals
         IF NOT #_ciReq[#_i] THEN
           #Diag.Station[#_i].CheckIn.UnexpectedDone := TRUE;
         END_IF;
       END_IF;
       #_ciDonePrev[#_i] := #_ciDone[#_i];

       // Add to totals (totals are sum of per-station counters)
       #Diag.Counters.TotalDone_CheckIn := #Diag.Counters.TotalDone_CheckIn + #Diag.Station[#_i].CheckIn.CountDone;
       #Diag.Counters.TotalTimeout_CheckIn := #Diag.Counters.TotalTimeout_CheckIn + #Diag.Station[#_i].CheckIn.CountTimeout;
       #Diag.Counters.TotalOK_CheckIn := #Diag.Counters.TotalOK_CheckIn + #Diag.Station[#_i].CheckIn.CountOK;
       #Diag.Counters.TotalNG_CheckIn := #Diag.Counters.TotalNG_CheckIn + #Diag.Station[#_i].CheckIn.CountNG;


       // --------------------------------------------------------------------------
       // CHECK-OUT DIAG (Unload)
       // --------------------------------------------------------------------------
       #Diag.Station[#_i].CheckOut.Req := #_coReq[#_i];
       #Diag.Station[#_i].CheckOut.StoredOK := #_coOk[#_i];
       #Diag.Station[#_i].CheckOut.StoredNG := #_coNg[#_i];
       #Diag.Station[#_i].CheckOut.Done := #_coDone[#_i];

       // Invalid state detector: OK and NG simultaneously
       #Diag.Station[#_i].CheckOut.BothOkNg := #_coOk[#_i] AND #_coNg[#_i];

       // Rising edge count: OK
       IF #_coOk[#_i] AND (NOT #_coOkPrev[#_i]) THEN
         #Diag.Station[#_i].CheckOut.CountOK := #Diag.Station[#_i].CheckOut.CountOK + 1;
       END_IF;
       #_coOkPrev[#_i] := #_coOk[#_i];

       // Rising edge count: NG
       IF #_coNg[#_i] AND (NOT #_coNgPrev[#_i]) THEN
         #Diag.Station[#_i].CheckOut.CountNG := #Diag.Station[#_i].CheckOut.CountNG + 1;
       END_IF;
       #_coNgPrev[#_i] := #_coNg[#_i];

       // Timer: measure duration of active request
       IF #_coReq[#_i] THEN
         #_tCo[#_i](IN := TRUE,
                    PT := #CheckOutTimeout);
         #Diag.Station[#_i].CheckOut.InProgress := TRUE;
       ELSE
         // Reset timer when request is inactive
         #_tCo[#_i](IN := FALSE,
                    PT := t#100ms);
         #Diag.Station[#_i].CheckOut.InProgress := FALSE;
       END_IF;

       #Diag.Station[#_i].CheckOut.Elapsed := #_tCo[#_i].ET;

       // Timeout: timer expired while request still active and Done not received
       #Diag.Station[#_i].CheckOut.Timeout :=
       #_tCo[#_i].Q AND #_coReq[#_i] AND (NOT #_coDone[#_i]);

       // Count timeout only once per timeout episode (latch)
       IF #Diag.Station[#_i].CheckOut.Timeout AND (NOT #_coTimeoutLatched[#_i]) THEN
         #_coTimeoutLatched[#_i] := TRUE;
         #Diag.Station[#_i].CheckOut.CountTimeout := #Diag.Station[#_i].CheckOut.CountTimeout + 1;
       END_IF;

       // Release latch when timeout clears
       IF NOT #Diag.Station[#_i].CheckOut.Timeout THEN
         #_coTimeoutLatched[#_i] := FALSE;
       END_IF;

       // Rising edge count: Done + UnexpectedDone latch if no active request
       IF #_coDone[#_i] AND (NOT #_coDonePrev[#_i]) THEN
         #Diag.Station[#_i].CheckOut.CountDone := #Diag.Station[#_i].CheckOut.CountDone + 1;

         // Done without request: indicates inconsistent handshake timing or stale signals
         IF NOT #_coReq[#_i] THEN
           #Diag.Station[#_i].CheckOut.UnexpectedDone := TRUE;
         END_IF;
       END_IF;
       #_coDonePrev[#_i] := #_coDone[#_i];

       // Add to totals
       #Diag.Counters.TotalDone_CheckOut := #Diag.Counters.TotalDone_CheckOut + #Diag.Station[#_i].CheckOut.CountDone;
       #Diag.Counters.TotalTimeout_CheckOut := #Diag.Counters.TotalTimeout_CheckOut + #Diag.Station[#_i].CheckOut.CountTimeout;
       #Diag.Counters.TotalOK_CheckOut := #Diag.Counters.TotalOK_CheckOut + #Diag.Station[#_i].CheckOut.CountOK;
       #Diag.Counters.TotalNG_CheckOut := #Diag.Counters.TotalNG_CheckOut + #Diag.Station[#_i].CheckOut.CountNG;


       // --------------------------------------------------------------------------
       // SUBPART DIAG (MES classification for subparts)
       // --------------------------------------------------------------------------
       #Diag.Station[#_i].SubPart.OK := #_spOk[#_i];
       #Diag.Station[#_i].SubPart.NG := #_spNg[#_i];
       #Diag.Station[#_i].SubPart.Done := #_spDone[#_i];

       #Diag.Station[#_i].SubPart.BothOkNg := #_spOk[#_i] AND #_spNg[#_i];

       // Rising edge count: OK
       IF #_spOk[#_i] AND (NOT #_spOkPrev[#_i]) THEN
         #Diag.Station[#_i].SubPart.CountOK := #Diag.Station[#_i].SubPart.CountOK + 1;
       END_IF;
       #_spOkPrev[#_i] := #_spOk[#_i];

       // Rising edge count: NG
       IF #_spNg[#_i] AND (NOT #_spNgPrev[#_i]) THEN
         #Diag.Station[#_i].SubPart.CountNG := #Diag.Station[#_i].SubPart.CountNG + 1;
       END_IF;
       #_spNgPrev[#_i] := #_spNg[#_i];

       // Rising edge count: Done
       IF #_spDone[#_i] AND (NOT #_spDonePrev[#_i]) THEN
         #Diag.Station[#_i].SubPart.CountDone := #Diag.Station[#_i].SubPart.CountDone + 1;
       END_IF;
       #_spDonePrev[#_i] := #_spDone[#_i];


       // --------------------------------------------------------------------------
       // LOAD RESULTS STORED DIAG (MES confirm storing results for load side)
       // --------------------------------------------------------------------------
       #Diag.Station[#_i].LoadResultsStored.OK := #_lrOk[#_i];
       #Diag.Station[#_i].LoadResultsStored.NG := #_lrNg[#_i];
       #Diag.Station[#_i].LoadResultsStored.Done := #_lrDone[#_i];

       #Diag.Station[#_i].LoadResultsStored.BothOkNg := #_lrOk[#_i] AND #_lrNg[#_i];

       // Rising edge count: OK
       IF #_lrOk[#_i] AND (NOT #_lrOkPrev[#_i]) THEN
         #Diag.Station[#_i].LoadResultsStored.CountOK := #Diag.Station[#_i].LoadResultsStored.CountOK + 1;
       END_IF;
       #_lrOkPrev[#_i] := #_lrOk[#_i];

       // Rising edge count: NG
       IF #_lrNg[#_i] AND (NOT #_lrNgPrev[#_i]) THEN
         #Diag.Station[#_i].LoadResultsStored.CountNG := #Diag.Station[#_i].LoadResultsStored.CountNG + 1;
       END_IF;
       #_lrNgPrev[#_i] := #_lrNg[#_i];

       // Rising edge count: Done
       IF #_lrDone[#_i] AND (NOT #_lrDonePrev[#_i]) THEN
         #Diag.Station[#_i].LoadResultsStored.CountDone := #Diag.Station[#_i].LoadResultsStored.CountDone + 1;
       END_IF;
       #_lrDonePrev[#_i] := #_lrDone[#_i];

     END_FOR;
   END_REGION


   REGION "SPECIAL HANDSHAKE - STOVE CHECK-IN (LOAD)"
     #Diag.Special.StoveCheckInReq := #_stoveReq;
     #Diag.Special.StoveCheckInOk := #_stoveOk;
     #Diag.Special.InProgress := #_stoveReq;

     // Timer runs while request active
     #_tStove(IN := #_stoveReq,
              PT := #StoveCheckInTimeout);

     #Diag.Special.Elapsed := #_tStove.ET;

     // Timeout: PT elapsed and still no OK
     #Diag.Special.Timeout := #_tStove.Q AND #_stoveReq AND (NOT #_stoveOk);

     // Rising edge count: OK
     IF #_stoveOk AND (NOT #_stoveOkPrev) THEN
       #Diag.Special.CountOk := #Diag.Special.CountOk + 1;
     END_IF;
     #_stoveOkPrev := #_stoveOk;

     // Count timeout only once per timeout episode
     IF #Diag.Special.Timeout AND (NOT #_stoveTimeoutLatched) THEN
       #_stoveTimeoutLatched := TRUE;
       #Diag.Special.CountTimeout := #Diag.Special.CountTimeout + 1;
     END_IF;

     IF NOT #Diag.Special.Timeout THEN
       #_stoveTimeoutLatched := FALSE;
     END_IF;
   END_REGION
END_FUNCTION_BLOCK
